KUKA KRL program: song_3.src, SONG_3.dat

--- song_3.src ---
&ACCESS RVO
&REL 22
&PARAM DISKPATH = KRC:\R1\Program\_KLAVIRISTA_V2\subprogram
DEF  SONG_3 ( )
;FOLD INI;%{PE}
  ;FOLD BASISTECH INI
    GLOBAL INTERRUPT DECL 3 WHEN $STOPMESS==TRUE DO IR_STOPM ( )
    INTERRUPT ON 3
    BAS (#INITMOV,0 )
  ;ENDFOLD (BASISTECH INI)
  ;FOLD USER INI
    ;Make your modifications here
INTERRUPT DECL 10 WHEN $IN[8] DO STOP_SONG()
INTERRUPT ON 10
INTERRUPT OFF 12
  ;ENDFOLD (USER INI)
;ENDFOLD (INI)
PIANO_ON_OFF()
IF PyMAX_VOLUME THEN
 VOLUME_MAX()
 ENDIF
;FOLD Otoceni koleckem
;FOLD PTP P14 Vel=17 % PDAT5 Tool[4]:TQGripper Base[1]:Piano ;%{PE}
;FOLD Parameters ;%{h}
;Params IlfProvider=kukaroboter.basistech.inlineforms.movement.old; Kuka.IsGlobalPoint=False; Kuka.PointName=P14; Kuka.BlendingEnabled=False; Kuka.MoveDataPtpName=PDAT5; Kuka.VelocityPtp=17; Kuka.CurrentCDSetIndex=0; Kuka.MovementParameterFieldEnabled=True; IlfCommand=PTP
;ENDFOLD
$BWDSTART = FALSE
PDAT_ACT = PPDAT5
FDAT_ACT = FP14
BAS(#PTP_PARAMS, 17.0)
SET_CD_PARAMS (0)
;PTP XP14
;ENDFOLD
;FOLD PTP P13 Vel=17 % PDAT4 Tool[4]:TQGripper Base[1]:Piano ;%{PE}
;FOLD Parameters ;%{h}
;Params IlfProvider=kukaroboter.basistech.inlineforms.movement.old; Kuka.IsGlobalPoint=False; Kuka.PointName=P13; Kuka.BlendingEnabled=False; Kuka.MoveDataPtpName=PDAT4; Kuka.VelocityPtp=17; Kuka.CurrentCDSetIndex=0; Kuka.MovementParameterFieldEnabled=True; IlfCommand=PTP
;ENDFOLD
$BWDSTART = FALSE
PDAT_ACT = PPDAT4
FDAT_ACT = FP13
BAS(#PTP_PARAMS, 17.0)
SET_CD_PARAMS (0)
;PTP XP13
;ENDFOLD
;FOLD PTP P9 Vel=17 % PDAT3 Tool[4]:TQGripper Base[1]:Piano ;%{PE}
;FOLD Parameters ;%{h}
;Params IlfProvider=kukaroboter.basistech.inlineforms.movement.old; Kuka.IsGlobalPoint=False; Kuka.PointName=P9; Kuka.BlendingEnabled=False; Kuka.MoveDataPtpName=PDAT3; Kuka.VelocityPtp=17; Kuka.CurrentCDSetIndex=0; Kuka.MovementParameterFieldEnabled=True; IlfCommand=PTP
;ENDFOLD
$BWDSTART = FALSE
PDAT_ACT = PPDAT3
FDAT_ACT = FP9
BAS(#PTP_PARAMS, 17.0)
SET_CD_PARAMS (0)
;PTP XP9
;ENDFOLD
;FOLD CIRC P10 P11 Vel=2 m/s CPDAT4 Tool[4]:TQGripper Base[1]:Piano ;%{PE}
;FOLD Parameters ;%{h}
;Params IlfProvider=kukaroboter.basistech.inlineforms.movement.old; Kuka.IsGlobalPoint=False; Kuka.PointName=P11; Kuka.HelpPointName=P10; Kuka.BlendingEnabled=False; Kuka.MoveDataName=CPDAT4; Kuka.VelocityPath=2; Kuka.CurrentCDSetIndex=0; Kuka.MovementParameterFieldEnabled=True; IlfCommand=CIRC
;ENDFOLD
$BWDSTART = FALSE
LDAT_ACT = LCPDAT4
FDAT_ACT = FP11
BAS(#CP_PARAMS, 2.0)
SET_CD_PARAMS (0)
;CIRC XP10, XP11
;ENDFOLD
;FOLD CIRC P12 P9 Vel=2 m/s CPDAT5 Tool[4]:TQGripper Base[1]:Piano ;%{PE}
;FOLD Parameters ;%{h}
;Params IlfProvider=kukaroboter.basistech.inlineforms.movement.old; Kuka.IsGlobalPoint=False; Kuka.PointName=P9; Kuka.HelpPointName=P12; Kuka.BlendingEnabled=False; Kuka.MoveDataName=CPDAT5; Kuka.VelocityPath=2; Kuka.CurrentCDSetIndex=0; Kuka.MovementParameterFieldEnabled=True; IlfCommand=CIRC
;ENDFOLD
$BWDSTART = FALSE
LDAT_ACT = LCPDAT5
FDAT_ACT = FP9
BAS(#CP_PARAMS, 2.0)
SET_CD_PARAMS (0)
;CIRC XP12, XP9
;ENDFOLD
;FOLD PTP P14 Vel=17 % PDAT5 Tool[4]:TQGripper Base[1]:Piano ;%{PE}
;FOLD Parameters ;%{h}
;Params IlfProvider=kukaroboter.basistech.inlineforms.movement.old; Kuka.IsGlobalPoint=False; Kuka.PointName=P14; Kuka.BlendingEnabled=False; Kuka.MoveDataPtpName=PDAT5; Kuka.VelocityPtp=17; Kuka.CurrentCDSetIndex=0; Kuka.MovementParameterFieldEnabled=True; IlfCommand=PTP
;ENDFOLD
$BWDSTART = FALSE
PDAT_ACT = PPDAT5
FDAT_ACT = FP14
BAS(#PTP_PARAMS, 17.0)
SET_CD_PARAMS (0)
;PTP XP14
;ENDFOLD
;ENDFOLD
SUSTAIN_ON_OFF()
BAR = 600
GRIPPER(2,TRUE)
GRIPPER(3,FALSE)
PLAY(9,0,0.5*BAR)
PLAY(9,0,0.5*BAR)
PLAY(10,0,0.5*BAR)
PLAY(11,0,0.5*BAR)
PLAY(11,0,0.5*BAR)
PLAY(10,0,0.5*BAR)
PLAY(9,0,0.5*BAR)
GRIPPER(4,FALSE)
PLAY(7.5,0,0.75*BAR)

PLAY(6.5,0,0.5*BAR)
PLAY(6.5,0,0.5*BAR)
GRIPPER(3,FALSE)
PLAY(8,0,0.5*BAR)
PLAY(9,0,0.5*BAR)
PLAY(9,0,0.75*BAR)
PLAY(8,0,0.25*BAR)
PLAY(8,0,2*BAR)


PLAY(9,0,0.5*BAR)
PLAY(9,0,0.5*BAR)
PLAY(10,0,0.5*BAR)
PLAY(11,0,0.5*BAR)
PLAY(11,0,0.5*BAR)
PLAY(10,0,0.5*BAR)
PLAY(9,0,0.5*BAR)
GRIPPER(4,FALSE)
PLAY(7.5,0,0.75*BAR)

PLAY(6.5,0,0.5*BAR)
PLAY(6.5,0,0.5*BAR)
GRIPPER(3,FALSE)
PLAY(8,0,0.5*BAR)
PLAY(9,0,0.5*BAR)
PLAY(8,0,0.75*BAR)
GRIPPER(4,FALSE)
PLAY(6.5,0,0.25*BAR)
PLAY(6.5,0,2*BAR)

GRIPPER(3,TRUE)
GRIPPER(2,TRUE)
GRIPPER(1,TRUE)

PIANO_ON_OFF()
;FOLD PyEND reset
PyEND = TRUE
Wait sec 0.2
PyEND = FALSE
;ENDFOLD
END

--- SONG_3.dat ---
&ACCESS RVO
&REL 22
&PARAM DISKPATH = KRC:\R1\Program\_KLAVIRISTA_V2\subprogram
DEFDAT  SONG_3
;FOLD EXTERNAL DECLARATIONS;%{PE}%MKUKATPBASIS,%CEXT,%VCOMMON,%P
;FOLD BASISTECH EXT;%{PE}%MKUKATPBASIS,%CEXT,%VEXT,%P
EXT  BAS (BAS_COMMAND  :IN,REAL  :IN )
DECL INT COUNT
DECL INT BAR
DECL REAL vysledek
;ENDFOLD (BASISTECH EXT)
;FOLD USER EXT;%{E}%MKUKATPUSER,%CEXT,%VEXT,%P
;Make your modifications here

;ENDFOLD (USER EXT)
;ENDFOLD (EXTERNAL DECLARATIONS)
DECL E6POS XP1={X 254.074,Y -71.6057739,Z 428.638428,A 11.2668905,B 14.5052948,C -177.268250,S 2,T 2,E1 0.0,E2 0.0,E3 0.0,E4 0.0,E5 0.0,E6 0.0}
DECL FDAT FP1={TOOL_NO 1,BASE_NO 0,IPO_FRAME #BASE,POINT2[] " "}
DECL PDAT PPDAT1={VEL 100.000,ACC 100.000,APO_DIST 500.000,APO_MODE #CDIS,GEAR_JERK 100.000,EXAX_IGN 0}
DECL MODULEPARAM_T LAST_TP_PARAMS={PARAMS[] "Kuka.PointName=P14; Kuka.FrameData.base_no=1; Kuka.FrameData.tool_no=4; Kuka.FrameData.ipo_frame=#BASE; Kuka.isglobalpoint=False; Kuka.MoveDataPtpName=PDAT5; Kuka.MovementDataPdat.apo_mode=#CDIS; Kuka.MovementDataPdat.apo_dist=500; Kuka.MovementData.vel=17; Kuka.MovementData.acc=100; Kuka.MovementData.exax_ign=0; Kuka.VelocityPtp=17; Kuka.BlendingEnabled=False; Kuka.APXEnabled=False; Kuka.CurrentCDSetIndex=0; Kuka.MoveDataName=CPDAT5; Kuka.MovementData.apo_fac=50; Kuka.MovementData.apo_dist=500; Kuka.MovementData.axis_acc=100; Kuka.MovementData.axis_vel=100; Kuka.MovementData.circ_typ=#BASE; Kuka.MovementData.jerk_fac=50; Kuka.MovementData.ori_typ=#VAR; Kuka.VelocityPath=2; Kuka.HelpPointName=P12; Kuka.FrameData.point2=      "}
DECL E6POS XP2={X 261.830963,Y -62.2262535,Z 427.296844,A 11.1519966,B 14.5930262,C -177.725601,S 2,T 2,E1 0.0,E2 0.0,E3 0.0,E4 0.0,E5 0.0,E6 0.0}
DECL E6POS XP3={X 268.946136,Y -70.7355576,Z 426.451691,A 11.0334129,B 14.3070974,C -177.815292,S 2,T 2,E1 0.0,E2 0.0,E3 0.0,E4 0.0,E5 0.0,E6 0.0}
DECL FDAT FP3={TOOL_NO 1,BASE_NO 0,IPO_FRAME #BASE,POINT2[] " "}
DECL LDAT LCPDAT1={VEL 2.00000,ACC 100.000,APO_DIST 500.000,APO_FAC 50.0000,AXIS_VEL 100.000,AXIS_ACC 100.000,ORI_TYP #VAR,CIRC_TYP #BASE,JERK_FAC 50.0000,GEAR_JERK 100.000,EXAX_IGN 0}
DECL E6POS XP4={X 261.090698,Y -78.9066544,Z 427.396240,A 11.0420723,B 14.3005857,C -177.780579,S 2,T 2,E1 0.0,E2 0.0,E3 0.0,E4 0.0,E5 0.0,E6 0.0}
DECL E6POS XP5={X 253.729904,Y -70.4463196,Z 428.379272,A 11.0482178,B 14.2959480,C -177.755890,S 2,T 2,E1 0.0,E2 0.0,E3 0.0,E4 0.0,E5 0.0,E6 0.0}
DECL FDAT FP5={TOOL_NO 1,BASE_NO 0,IPO_FRAME #BASE,POINT2[] " "}
DECL LDAT LCPDAT2={VEL 2.00000,ACC 100.000,APO_DIST 500.000,APO_FAC 50.0000,AXIS_VEL 100.000,AXIS_ACC 100.000,ORI_TYP #VAR,CIRC_TYP #BASE,JERK_FAC 50.0000,GEAR_JERK 100.000,EXAX_IGN 0}
DECL E6POS XP7={X 253.729904,Y -70.4463196,Z 428.379272,A 11.0482178,B 14.2959480,C -177.755890,S 2,T 2,E1 0.0,E2 0.0,E3 0.0,E4 0.0,E5 0.0,E6 0.0}
DECL E6POS XP6={X 261.090698,Y -78.9066544,Z 427.396240,A 11.0420723,B 14.3005857,C -177.780579,S 2,T 2,E1 0.0,E2 0.0,E3 0.0,E4 0.0,E5 0.0,E6 0.0}
DECL FDAT FP7={TOOL_NO 1,BASE_NO 0,IPO_FRAME #BASE,POINT2[] " "}
DECL LDAT LCPDAT3={VEL 2.00000,ACC 100.000,APO_DIST 500.000,APO_FAC 50.0000,AXIS_VEL 100.000,AXIS_ACC 100.000,ORI_TYP #VAR,CIRC_TYP #BASE,JERK_FAC 50.0000,GEAR_JERK 100.000,EXAX_IGN 0}
DECL E6POS XP8={X 247.112442,Y -70.4753342,Z 450.676422,A 10.8469791,B 10.0203524,C -178.609650,S 2,T 2,E1 0.0,E2 0.0,E3 0.0,E4 0.0,E5 0.0,E6 0.0}
DECL FDAT FP8={TOOL_NO 1,BASE_NO 0,IPO_FRAME #BASE,POINT2[] " "}
DECL PDAT PPDAT2={VEL 17.0000,ACC 100.000,APO_DIST 500.000,APO_MODE #CDIS,GEAR_JERK 100.000,EXAX_IGN 0}
DECL E6POS XP9={X 172.905655,Y 181.593323,Z 25.3962860,A -79.3194733,B 14.3763237,C -177.332870,S 2,T 2,E1 0.0,E2 0.0,E3 0.0,E4 0.0,E5 0.0,E6 0.0}
DECL FDAT FP9={TOOL_NO 4,BASE_NO 1,IPO_FRAME #BASE,POINT2[] " "}
DECL PDAT PPDAT3={VEL 17.0000,ACC 100.000,APO_DIST 500.000,APO_MODE #CDIS,GEAR_JERK 100.000,EXAX_IGN 0}
DECL E6POS XP10={X 181.839462,Y 174.177444,Z 25.2611942,A -79.3199463,B 14.3775740,C -177.339371,S 2,T 2,E1 0.0,E2 0.0,E3 0.0,E4 0.0,E5 0.0,E6 0.0}
DECL E6POS XP11={X 174.167816,Y 165.910507,Z 23.0958385,A -79.3199463,B 14.3775740,C -177.339371,S 2,T 2,E1 0.0,E2 0.0,E3 0.0,E4 0.0,E5 0.0,E6 0.0}
DECL FDAT FP11={TOOL_NO 4,BASE_NO 1,IPO_FRAME #BASE,POINT2[] " "}
DECL LDAT LCPDAT4={VEL 2.00000,ACC 100.000,APO_DIST 500.000,APO_FAC 50.0000,AXIS_VEL 100.000,AXIS_ACC 100.000,ORI_TYP #VAR,CIRC_TYP #BASE,JERK_FAC 50.0000,GEAR_JERK 100.000,EXAX_IGN 0}
DECL E6POS XP12={X 165.340317,Y 173.766632,Z 24.5302486,A -79.3198776,B 14.3775167,C -177.339081,S 2,T 2,E1 0.0,E2 0.0,E3 0.0,E4 0.0,E5 0.0,E6 0.0}
DECL LDAT LCPDAT5={VEL 2.00000,ACC 100.000,APO_DIST 500.000,APO_FAC 50.0000,AXIS_VEL 100.000,AXIS_ACC 100.000,ORI_TYP #VAR,CIRC_TYP #BASE,JERK_FAC 50.0000,GEAR_JERK 100.000,EXAX_IGN 0}
DECL E6POS XP13={X 173.818314,Y 178.829681,Z 48.7109146,A -79.6227341,B 11.1214085,C -178.258255,S 2,T 2,E1 0.0,E2 0.0,E3 0.0,E4 0.0,E5 0.0,E6 0.0}
DECL FDAT FP13={TOOL_NO 4,BASE_NO 1,IPO_FRAME #BASE,POINT2[] " "}
DECL PDAT PPDAT4={VEL 17.0000,ACC 100.000,APO_DIST 500.000,APO_MODE #CDIS,GEAR_JERK 100.000,EXAX_IGN 0}
DECL E6POS XP14={X 173.818314,Y 178.829681,Z 48.7109146,A -79.6227341,B 11.1214085,C -178.258255,S 2,T 2,E1 0.0,E2 0.0,E3 0.0,E4 0.0,E5 0.0,E6 0.0}
DECL FDAT FP14={TOOL_NO 4,BASE_NO 1,IPO_FRAME #BASE,POINT2[] " "}
DECL PDAT PPDAT5={VEL 17.0000,ACC 100.000,APO_DIST 500.000,APO_MODE #CDIS,GEAR_JERK 100.000,EXAX_IGN 0}
ENDDAT
